// TIA Portal V19 export
DATA_BLOCK "DecoilersHU"   // DB61
// stored: InstanceOfName DecoilersHU_FB, InstanceOfType FB
"DecoilersHU_FB"
   // VAR_INPUT
   //    AreaInterface : "AreaInterface";
   //    ZSI : "udt_ZoneSafetyInterface";
   //    DSI : "udt_DeviceSafetyInterface";
   //    DataIn : Struct
   //       Pb_Stop : Bool;
   //       Pb_Start : Bool;
   //    END_STRUCT;
   //    CIn : Struct
   //       EnableStopStopDueDoorOpeningRequest : Bool;
   //       EnableStopInPhase : Bool;
   //       EnableStopProgrammed : Bool;
   //       PressureReq : Bool;
   //    END_STRUCT;
   // END_VAR
   // VAR_OUTPUT
   //    MachineInterface : "MachineInterface";
   //    DataOut : Struct
   //       Pressure_V : Bool;
   //    END_STRUCT;
   //    COut : Struct
   //       Standstill : Bool;
   //       Run_CheckNext : Bool;
   //       CtrlSafe : Bool;
   //       PressureRunning : Bool;
   //    END_STRUCT;
   // END_VAR
   // VAR
   //    Sts : Struct
   //       Standstill : Bool;
   //       AlarmsPresence : Bool;
   //       WarningsPresence : Bool;
   //       Cnd : Bool;
   //    END_STRUCT;
   //    Ctrl : Struct
   //       StopDueDoorOpeningRequest : Bool;
   //       StopInPhase : Bool;
   //       StopProgrammed : Bool;
   //       StopAborting : Bool;
   //       Run : Bool;
   //       Run_Man : Bool;
   //       Run_Aut : Bool;
   //    END_STRUCT;
   //    Alarm : Struct
   //       Pump : "MotorAlr";
   //    END_STRUCT;
   //    Warning : Struct
   //       NotAutReady : Bool;
   //    END_STRUCT;
   //    Pump_M : "Motor";
   //    TON_NoPendingCmd : IEC_TIMER;
   //    TON_Inactivity : IEC_TIMER;
   //    TON_Pressure { S7_SetPoint := 'True'} : IEC_TIMER;
   //    Aux : Struct
   //       Pb_Start : Bool;
   //    END_STRUCT;
   // END_VAR
BEGIN
END_DATA_BLOCK
